TYPE ST_AnalogLamp_fb :
STRUCT
	status: BOOL;
	brightness: INT;
	colorSelected: UDINT;
	errorID: UDINT;
END_STRUCT
END_TYPE

(* stored: Version 1.1.0.1, ProductVersion 3.1.4024.12
   DUT ST_AnalogLamp_fb: Id {d6c7d7f9-a665-4ddf-a829-7cf35451b276} *)
